TYPE ST_Data_PCR :
STRUCT
	dateTime			: STRING;
	pumpNo				: STRING;
	step				: STRING;
	tareWt				: STRING;
	grossWt				: STRING;
	netVolume			: STRING;
	netWt				: STRING;
	targetVolume		: STRING;
	differencePercent	: STRING;
	criteria			: STRING;
	pumpRevs			: STRING;
	CalibrationNo		: INT;
	
END_STRUCT
END_TYPE

(* stored: Version 1.1.0.1, ProductVersion 3.1.4024.15
   DUT ST_Data_PCR: Id {8041bc92-21c9-4be0-bdeb-d07fbadba5e3} *)
